FUNCTION F_LIMIT : BOOL
VAR_INPUT
	En			: BOOL;
	High		: LREAL;
	Value		: LREAL;
	Low			: LREAL;
END_VAR
VAR
END_VAR

IF En = TRUE AND (Low <= High AND
 (Value >= Low AND Value <= High)) OR
 (Low >= High AND
 (Value <= Low OR Value >= High)) THEN
	F_LIMIT := TRUE;
ELSE	
	F_LIMIT := FALSE;
END_IF;

END_FUNCTION

(* stored: Version 1.1.0.1, ProductVersion 3.1.4022.6
   POU F_LIMIT: Id {75ba2409-0d37-4166-b972-c727bfac775e}, SpecialFunc None *)
